FUNCTION TryConvert_DWORD_TO_WORD : BOOL
VAR_INPUT
	in : DWORD;
	out : REFERENCE TO WORD;
END_VAR

IF in > DatatypeLimits.MAX_VALUE_OF_DWORD_WHICH_CAN_BE_HELD_IN_A_WORD THEN
	RETURN;
END_IF

out := DWORD_TO_WORD(in);
TryConvert_DWORD_TO_WORD := TRUE;

END_FUNCTION

(* stored: Version 1.1.0.1, ProductVersion 3.1.4024.12
   POU TryConvert_DWORD_TO_WORD: Id {fd4e63d5-7e91-4569-8a4d-004e940a057a}, SpecialFunc None *)
